Universal Robots PolyScope program: ATI_example_SurfaceSearchandProcess.urp

Program ATI_example_SurfaceSearchandProcess_FIXED (createdIn=3.1.18024.0 lastSavedIn=5.0.0.30136 robotSerialNumber=2014309999 directory=/home/ur/ursim-current/programs/UR/DemoPrograms installation=default)
Calibrated DH parameters: a=[-0.000069, -0.581857, -0.429354, 0.000018, -0.000012, 0]; d=[0.18099, 126.33209, 113.191346, -239.349299, 0.119939, 0.115552]; alpha=[1.570758, -0.001509, -0.001573, 1.570435, -1.570714, 0]; deltaTheta=[0, -0.316668, 5.879502, 0.720355, -0.000001, 0]
BeforeStart
  Folder Move to Initial start position
    'Set Actual Robot Payload (enter your TCP payload)'
    Script: set_payload(1)
    'Move to a Start Position (reteach this point to a safe home location!)'
    MoveJ speed 60 deg/s, acceleration 80 deg/s^2 (useActiveTCP=false)
      Waypoint Start: TCP in base x=73.32 y=-708.856 z=677.514 mm, rx=-0.5453 ry=3.0922 rz=0.0003 rad; joints [-70.001, -89.997, -90, -90.004, 90.001, -0.002] deg
    Wait Sleep waitTime=0.01
    URCap F/T Sensor Options (ATI Axia Force/Torque Sensor, ATI Industrial Automation) dataModel(LOGGING_LEVEL=0, STATUS=80000008)
    URCap F/T Sensor Command (ATI Axia Force/Torque Sensor, ATI Industrial Automation) dataModel(running=Enable, WEIGHT=0.025)
    'Adjust sensitivity of UR Force mode'
    Script: force_mode_set_damping(1)
    Script: force_mode_set_gain_scaling(.5)
Robot Program (runOnlyOnce=true speed=0 acceleration=0 useActiveTCP=false) feature=Base
  Folder Bias the sensor
    Wait Sleep waitTime=1
    URCap F/T Sensor Command (ATI Axia Force/Torque Sensor, ATI Industrial Automation) dataModel(running=Bias)
  Folder Move down until the tool touches a surface
    MoveJ speed 60 deg/s, acceleration 80 deg/s^2 (useActiveTCP=true)
      'Move to hover above surface (reteach to a point ~5cm above surface)'
      Waypoint AboveTable: TCP in base x=73.483 y=-708.833 z=280.453 mm, rx=-0.5454 ry=3.0923 rz=0.0003 rad; joints [-69.997, -97.634, -113.303, -59.062, 90.027, -0.032] deg; TCP offset x=0 y=0 z=98 mm, rx=0 ry=0 rz=0 rad
    If ATI_ZForce>-2 (checkContinuously=true)
      'Relative motion in Z'
      Script: movel(pose_trans(get_actual_tcp_pose(),p[0,0,.2,0,0,0]),a=0.05,v=.04,t=0,r=0)
  Folder Move across the surface while applying 2N of force
    Force Simple feature=Joint_6_name; selection=[0, 0, 1, 0, 0, 0]; wrench=[0, 0, 2, 0, 0, 0]; limitsForce=[0.15, 0.15, 0.15, 1.047198, 1.047198, 1.047198]; limitsMotion=[0.1, 0.1, 0.1, 0.349066, 0.349066, 0.349066]
      Folder If the tool encounters too much resistance, return to start position
        If xyPlaneForce <20 (checkContinuously=true)
          'Relative motion 0.3m in -Y'
          Script: movel(pose_trans(get_actual_tcp_pose(), p[0,-.3,0,0,0,0]),a=0.04,v=.02,t=0,r=0)
  Folder Reset to a start position
    'Relative motion in Z'
    Script: movel(pose_trans(get_actual_tcp_pose(), p[0,0,-.2,0,0,0]),a=0.04,v=.1,t=0,r=0)
  Folder Move down until the tool touchs a surface
    If ATI_ZForce>-2 (checkContinuously=true)
      'Relative motion in Z'
      Script: movel(pose_trans(get_actual_tcp_pose(),p[0,0,.2,0,0,0]),a=0.05,v=.04,t=0,r=0)
  Folder Move across the surface while applying 2N of force
    Force Simple feature=Joint_6_name; selection=[0, 0, 1, 0, 0, 0]; wrench=[0, 0, 2, 0, 0, 0]; limitsForce=[0.15, 0.15, 0.15, 1.047198, 1.047198, 1.047198]; limitsMotion=[0.1, 0.1, 0.1, 0.349066, 0.349066, 0.349066]
      Folder If the tool encounters too much resistance, return to start position
        If xyPlaneForce <20 (checkContinuously=true)
          'Relative motion 0.3m in +Y'
          Script: movel(pose_trans(get_actual_tcp_pose(), p[0,.3,0,0,0,0]),a=0.04,v=.02,t=0,r=0)
  Folder Reset to a start position
    Script: movel(pose_trans(get_actual_tcp_pose(), p[0,0,-.2,0,0,0]),a=0.04,v=.1,t=0,r=0)
    MoveJ speed 60 deg/s, acceleration 80 deg/s^2 (useActiveTCP=true)
      Waypoint Start: TCP in base x=73.32 y=-708.856 z=677.514 mm, rx=-0.5453 ry=3.0922 rz=0.0003 rad; joints [-70.001, -89.997, -90, -90.004, 90.001, -0.002] deg
Thread Thread_1 (runOnlyOnce=false trackProgramExecution=false)
  'UR Command get_tcp_force() is transformed to Base'
  TCPForce := get_tcp_force()
  'ATI reading in the sensor frame'
  ATI_rawFT := ati_ftsensor.get_raw_ft()
  'Adjust the TCP offset parameters for your tool!'
  'ATI reading in the TCP frame: TCP is .5 offset in Z from the sensor measuring face'
  ATI_TCP_FT := ati_ftsensor.get_tcp_ft(0, 0, .5, 0, 0, 0)
  ATI_ZForce := ATI_TCP_FT[2]
  Folder Get magnitude of force in X-Y plane, accounting for friction of tool
    xyPlaneForce := sqrt(pow(TCPForce[0], 2) + pow(TCPForce[1], 2)) - 0.3*ATI_ZForce
  Wait Sleep waitTime=0.01
